// TIA Portal V16 export
// export: Created 2022-11-01T21:54:10.387735Z, ExportSetting WithDefaults, DisplayName Totally Integrated Automation Portal, DisplayVersion V16, DisplayName TIA Portal Version Control Interface, DisplayVersion V16, DisplayName TIA Portal Openness, DisplayVersion V16, DisplayName SINAMICS Startdrive Advanced, DisplayVersion V16, DisplayName SINAMICS Startdrive G130, G150, S120, S150, SINAMICS MV, S210, DisplayVersion V16, DisplayName SINAMICS Startdrive G110M, G120, G120C, G120D, G120P, DisplayVersion V16, DisplayName STEP 7 Professional, DisplayVersion V16, DisplayName STEP 7 Safety, DisplayVersion V16, DisplayName WinCC Professional, DisplayVersion V16
VAR_GLOBAL   // PLC tag table "DI/O C500"
   "iH501/1_Run_Km" AT %M1700.0 : Bool;
   "iH501/1_Con_Vfd" AT %M1846.0 : Bool;
   "iH501/1_Run_Vfd" AT %M1846.1 : Bool;
   "qH501/1_Sel_Loc/Rem" AT %M1846.2 : Bool;
   "qH501/1_Sel_Km/Vfd" AT %M1846.3 : Bool;
   "qH501/1_Block" AT %M1846.4 : Bool;
   "qH501/1_Connect_Vfd" AT %M1846.5 : Bool;
   "qH501/1_Start" AT %M1846.6 : Bool;
   "iH501/2_Run_Km" AT %M1846.7 : Bool;
   "iH501/2_Con_Vfd" AT %M1847.0 : Bool;
   "iH501/2_Run_Vfd" AT %M1847.1 : Bool;
   "qH501/2_Sel_Loc/Rem" AT %M1847.2 : Bool;
   "qH501/2_Sel_Km/Vfd" AT %M1847.3 : Bool;
   "qH501/2_Block" AT %M1847.4 : Bool;
   "qH501/2_Connect_Vfd" AT %M1847.5 : Bool;
   "qH501/2_Start" AT %M1847.6 : Bool;
   "iH501/3_Run_Km" AT %M1847.7 : Bool;
   "iH501/3_Con_Vfd" AT %M1848.0 : Bool;
   "iH501/3_Run_Vfd" AT %M1848.1 : Bool;
   "qH501/3_Sel_Loc/Rem" AT %M1848.2 : Bool;
   "qH501/3_Sel_Km/Vfd" AT %M1848.3 : Bool;
   "qH501/3_Block" AT %M1848.4 : Bool;
   "qH501/3_Connect_Vfd" AT %M1848.5 : Bool;
   "qH501/3_Start" AT %M1848.6 : Bool;
   "iH501/4_Run_Km" AT %M1848.7 : Bool;
   "iH501/4_Con_Vfd" AT %M1849.0 : Bool;
   "iH501/4_Run_Vfd" AT %M1849.1 : Bool;
   "qH501/4_Sel_Loc/Rem" AT %M1849.2 : Bool;
   "qH501/4_Sel_Km/Vfd" AT %M1849.3 : Bool;
   "qH501/4_Block" AT %M1849.4 : Bool;
   "qH501/4_Connect_Vfd" AT %M1849.5 : Bool;
   "qH501/4_Start" AT %M1849.6 : Bool;
   "iH501/5_Run_Km" AT %M1849.7 : Bool;
   "iH501/5_Con_Vfd" AT %M1850.0 : Bool;
   "iH501/5_Run_Vfd" AT %M1850.1 : Bool;
   "qH501/5_Sel_Loc/Rem" AT %M1850.2 : Bool;
   "qH501/5_Sel_Km/Vfd" AT %M1850.3 : Bool;
   "qH501/5_Block" AT %M1850.4 : Bool;
   "qH501/5_Connect_Vfd" AT %M1850.5 : Bool;
   "qH501/5_Start" AT %M1850.6 : Bool;
   "iH502/1_Run_Km" AT %M1850.7 : Bool;
   "iH502/1_Con_Vfd" AT %M1851.0 : Bool;
   "iH502/1_Run_Vfd" AT %M1851.1 : Bool;
   "qH502/1_Sel_Loc/Rem" AT %M1851.2 : Bool;
   "qH502/1_Sel_Km/Vfd" AT %M1851.3 : Bool;
   "qH502/1_Block" AT %M1851.4 : Bool;
   "qH502/1_Connect_Vfd" AT %M1851.5 : Bool;
   "qH502/1_Start" AT %M1851.6 : Bool;
   "iH502/2_Run_Km" AT %M1851.7 : Bool;
   "iH502/2_Con_Vfd" AT %M1852.0 : Bool;
   "iH502/2_Run_Vfd" AT %M1852.1 : Bool;
   "qH502/2_Sel_Loc/Rem" AT %M1852.2 : Bool;
   "qH502/2_Sel_Km/Vfd" AT %M1852.3 : Bool;
   "qH502/2_Block" AT %M1852.4 : Bool;
   "qH502/2_Connect_Vfd" AT %M1852.5 : Bool;
   "qH502/2_Start" AT %M1852.6 : Bool;
   "iH502/3_Run_Km" AT %M1852.7 : Bool;
   "iH502/3_Con_Vfd" AT %M1853.0 : Bool;
   "iH502/3_Run_Vfd" AT %M1853.1 : Bool;
   "qH502/3_Sel_Loc/Rem" AT %M1853.2 : Bool;
   "qH502/3_Sel_Km/Vfd" AT %M1853.3 : Bool;
   "qH502/3_Block" AT %M1853.4 : Bool;
   "qH502/3_Connect_Vfd" AT %M1853.5 : Bool;
   "qH502/3_Start" AT %M1853.6 : Bool;
   "iH502/4_Run_Km" AT %M1853.7 : Bool;
   "iH502/4_Con_Vfd" AT %M1854.0 : Bool;
   "iH502/4_Run_Vfd" AT %M1854.1 : Bool;
   "qH502/4_Sel_Loc/Rem" AT %M1854.2 : Bool;
   "qH502/4_Sel_Km/Vfd" AT %M1854.3 : Bool;
   "qH502/4_Block" AT %M1854.4 : Bool;
   "qH502/4_Connect_Vfd" AT %M1854.5 : Bool;
   "qH502/4_Start" AT %M1854.6 : Bool;
   "iH502/5_Run_Km" AT %M1854.7 : Bool;
   "iH502/5_Con_Vfd" AT %M1855.0 : Bool;
   "iH502/5_Run_Vfd" AT %M1855.1 : Bool;
   "qH502/5_Sel_Loc/Rem" AT %M1855.2 : Bool;
   "qH502/5_Sel_Km/Vfd" AT %M1855.3 : Bool;
   "qH502/5_Block" AT %M1855.4 : Bool;
   "qH502/5_Connect_Vfd" AT %M1855.5 : Bool;
   "qH502/5_Start" AT %M1855.6 : Bool;
   "iH502/6_Run_Km" AT %M1855.7 : Bool;
   "iH502/6_Con_Vfd" AT %M1856.0 : Bool;
   "iH502/6_Run_Vfd" AT %M1856.1 : Bool;
   "qH502/6_Sel_Loc/Rem" AT %M1856.2 : Bool;
   "qH502/6_Sel_Km/Vfd" AT %M1856.3 : Bool;
   "qH502/6_Block" AT %M1856.4 : Bool;
   "qH502/6_Connect_Vfd" AT %M1856.5 : Bool;
   "qH502/6_Start" AT %M1856.6 : Bool;
   "iH502/7_Run_Km" AT %M1856.7 : Bool;
   "iH502/7_Con_Vfd" AT %M1857.0 : Bool;
   "iH502/7_Run_Vfd" AT %M1857.1 : Bool;
   "qH502/7_Sel_Loc/Rem" AT %M1857.2 : Bool;
   "qH502/7_Sel_Km/Vfd" AT %M1857.3 : Bool;
   "qH502/7_Block" AT %M1857.4 : Bool;
   "qH502/7_Connect_Vfd" AT %M1857.5 : Bool;
   "qH502/7_Start" AT %M1857.6 : Bool;
   "iH503/1_Run_Km" AT %M1857.7 : Bool;
   "iH503/1_Con_Vfd" AT %M1858.0 : Bool;
   "iH503/1_Run_Vfd" AT %M1858.1 : Bool;
   "qH503/1_Sel_Loc/Rem" AT %M1858.2 : Bool;
   "qH503/1_Sel_Km/Vfd" AT %M1858.3 : Bool;
   "qH503/1_Block" AT %M1858.4 : Bool;
   "qH503/1_Connect_Vfd" AT %M1858.5 : Bool;
   "qH503/1_Start" AT %M1858.6 : Bool;
   "iH503/2_Run_Km" AT %M1858.7 : Bool;
   "iH503/2_Con_Vfd" AT %M1859.0 : Bool;
   "iH503/2_Run_Vfd" AT %M1859.1 : Bool;
   "qH503/2_Sel_Loc/Rem" AT %M1859.2 : Bool;
   "qH503/2_Sel_Km/Vfd" AT %M1859.3 : Bool;
   "qH503/2_Block" AT %M1859.4 : Bool;
   "qH503/2_Connect_Vfd" AT %M1859.5 : Bool;
   "qH503/2_Start" AT %M1859.6 : Bool;
   "iH503/3_Run_Km" AT %M1859.7 : Bool;
   "iH503/3_Con_Vfd" AT %M1860.0 : Bool;
   "iH503/3_Run_Vfd" AT %M1860.1 : Bool;
   "qH503/3_Sel_Loc/Rem" AT %M1860.2 : Bool;
   "qH503/3_Sel_Km/Vfd" AT %M1860.3 : Bool;
   "qH503/3_Block" AT %M1860.4 : Bool;
   "qH503/3_Connect_Vfd" AT %M1860.5 : Bool;
   "qH503/3_Start" AT %M1860.6 : Bool;
   "iH503/4_Run_Km" AT %M1860.7 : Bool;
   "iH503/4_Con_Vfd" AT %M1861.0 : Bool;
   "iH503/4_Run_Vfd" AT %M1861.1 : Bool;
   "qH503/4_Sel_Loc/Rem" AT %M1861.2 : Bool;
   "qH503/4_Sel_Km/Vfd" AT %M1861.3 : Bool;
   "qH503/4_Block" AT %M1861.4 : Bool;
   "qH503/4_Connect_Vfd" AT %M1861.5 : Bool;
   "qH503/4_Start" AT %M1861.6 : Bool;
   "iH503/5_Run_Km" AT %M1861.7 : Bool;
   "iH503/5_Con_Vfd" AT %M1862.0 : Bool;
   "iH503/5_Run_Vfd" AT %M1862.1 : Bool;
   "qH503/5_Sel_Loc/Rem" AT %M1862.2 : Bool;
   "qH503/5_Sel_Km/Vfd" AT %M1862.3 : Bool;
   "qH503/5_Block" AT %M1862.4 : Bool;
   "qH503/5_Connect_Vfd" AT %M1862.5 : Bool;
   "qH503/5_Start" AT %M1862.6 : Bool;
   "iH503/6_Run_Km" AT %M1862.7 : Bool;
   "iH503/6_Con_Vfd" AT %M1863.0 : Bool;
   "iH503/6_Run_Vfd" AT %M1863.1 : Bool;
   "qH503/6_Sel_Loc/Rem" AT %M1863.2 : Bool;
   "qH503/6_Sel_Km/Vfd" AT %M1863.3 : Bool;
   "qH503/6_Block" AT %M1863.4 : Bool;
   "qH503/6_Connect_Vfd" AT %M1863.5 : Bool;
   "qH503/6_Start" AT %M1863.6 : Bool;
   "iH503/7_Run_Km" AT %M1863.7 : Bool;
   "iH503/7_Con_Vfd" AT %M1864.0 : Bool;
   "iH503/7_Run_Vfd" AT %M1864.1 : Bool;
   "qH503/7_Sel_Loc/Rem" AT %M1864.2 : Bool;
   "qH503/7_Sel_Km/Vfd" AT %M1864.3 : Bool;
   "qH503/7_Block" AT %M1864.4 : Bool;
   "qH503/7_Connect_Vfd" AT %M1864.5 : Bool;
   "qH503/7_Start" AT %M1864.6 : Bool;
   iUV501_Opn AT %M1864.7 : Bool;
   iUV501_Cls AT %M1865.0 : Bool;
   qUV501 AT %M1865.1 : Bool;
   "iH508/1_Run_Km" AT %M1865.2 : Bool;
   "iH508/1_Con_Vfd" AT %M1865.3 : Bool;
   "iH508/1_Run_Vfd" AT %M1865.4 : Bool;
   "qH508/1_Sel_Loc/Rem" AT %M1865.5 : Bool;
   "qH508/1_Sel_Km/Vfd" AT %M1865.6 : Bool;
   "qH508/1_Block" AT %M1865.7 : Bool;
   "qH508/1_Connect_Vfd" AT %M1876.0 : Bool;
   "qH508/1_Start" AT %M1876.1 : Bool;
   "iH508/2_Run_Km" AT %M1876.2 : Bool;
   "iH508/2_Con_Vfd" AT %M1876.3 : Bool;
   "iH508/2_Run_Vfd" AT %M1876.4 : Bool;
   "qH508/2_Sel_Loc/Rem" AT %M1876.5 : Bool;
   "qH508/2_Sel_Km/Vfd" AT %M1876.6 : Bool;
   "qH508/2_Block" AT %M1876.7 : Bool;
   "qH508/2_Connect_Vfd" AT %M1877.0 : Bool;
   "qH508/2_Start" AT %M1877.1 : Bool;
   "iH513/1_Run_Km" AT %M1877.2 : Bool;
   "iH513/1_Con_Vfd" AT %M1877.3 : Bool;
   "iH513/1_Run_Vfd" AT %M1877.4 : Bool;
   "qH513/1_Sel_Loc/Rem" AT %M1877.5 : Bool;
   "qH513/1_Sel_Km/Vfd" AT %M1877.6 : Bool;
   "qH513/1_Block" AT %M1877.7 : Bool;
   "qH513/1_Connect_Vfd" AT %M1878.0 : Bool;
   "qH513/1_Start" AT %M1878.1 : Bool;
   "iH513/2_Run_Km" AT %M1878.2 : Bool;
   "iH513/2_Con_Vfd" AT %M1878.3 : Bool;
   "iH513/2_Run_Vfd" AT %M1878.4 : Bool;
   "qH513/2_Sel_Loc/Rem" AT %M1878.5 : Bool;
   "qH513/2_Sel_Km/Vfd" AT %M1878.6 : Bool;
   "qH513/2_Block" AT %M1878.7 : Bool;
   "qH513/2_Connect_Vfd" AT %M1879.0 : Bool;
   "qH513/2_Start" AT %M1879.1 : Bool;
   iH507_Run_Km AT %M1879.2 : Bool;
   iH507_Con_Vfd AT %M1879.3 : Bool;
   iH507_Run_Vfd AT %M1879.4 : Bool;
   "qH507_Sel_Loc/Rem" AT %M1879.5 : Bool;
   "qH507_Sel_Km/Vfd" AT %M1879.6 : Bool;
   qH507_Block AT %M1879.7 : Bool;
   qH507_Connect_Vfd AT %M1880.0 : Bool;
   qH507_Start AT %M1880.1 : Bool;
END_VAR
